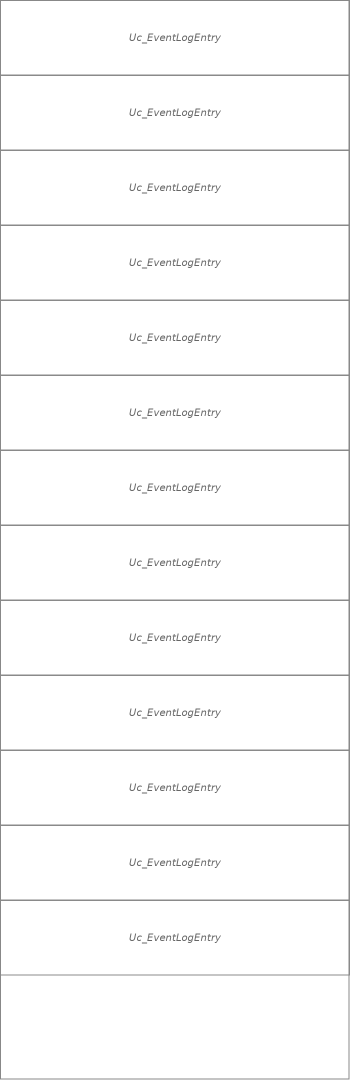
VISUALIZATION Uc_EventLogTable  // 350x1080
    Frame (0,0 350x75)
        shows Uc_EventLogEntry(stVisu := stVisu.astEvents[0], nSelectId := stVisu.nIdx, bQuit := stVisu.bQuitt)
    Frame (0,75 350x75)
        shows Uc_EventLogEntry(stVisu := stVisu.astEvents[1], nSelectId := stVisu.nIdx, bQuit := stVisu.bQuitt)
    Frame (0,150 350x75)
        shows Uc_EventLogEntry(stVisu := stVisu.astEvents[2], nSelectId := stVisu.nIdx, bQuit := stVisu.bQuitt)
    Frame (0,225 350x75)
        shows Uc_EventLogEntry(stVisu := stVisu.astEvents[3], nSelectId := stVisu.nIdx, bQuit := stVisu.bQuitt)
    Frame (0,300 350x75)
        shows Uc_EventLogEntry(stVisu := stVisu.astEvents[4], nSelectId := stVisu.nIdx, bQuit := stVisu.bQuitt)
    Frame (0,375 350x75)
        shows Uc_EventLogEntry(stVisu := stVisu.astEvents[5], nSelectId := stVisu.nIdx, bQuit := stVisu.bQuitt)
    Frame (0,450 350x75)
        shows Uc_EventLogEntry(stVisu := stVisu.astEvents[6], nSelectId := stVisu.nIdx, bQuit := stVisu.bQuitt)
    Frame (0,525 350x75)
        shows Uc_EventLogEntry(stVisu := stVisu.astEvents[7], nSelectId := stVisu.nIdx, bQuit := stVisu.bQuitt)
    Frame (0,600 350x75)
        shows Uc_EventLogEntry(stVisu := stVisu.astEvents[8], nSelectId := stVisu.nIdx, bQuit := stVisu.bQuitt)
    Frame (0,675 350x75)
        shows Uc_EventLogEntry(stVisu := stVisu.astEvents[9], nSelectId := stVisu.nIdx, bQuit := stVisu.bQuitt)
    Frame (0,750 350x75)
        shows Uc_EventLogEntry(stVisu := stVisu.astEvents[10], nSelectId := stVisu.nIdx, bQuit := stVisu.bQuitt)
    Frame (0,825 350x75)
        shows Uc_EventLogEntry(stVisu := stVisu.astEvents[11], nSelectId := stVisu.nIdx, bQuit := stVisu.bQuitt)
    Frame (0,900 350x75)
        shows Uc_EventLogEntry(stVisu := stVisu.astEvents[12], nSelectId := stVisu.nIdx, bQuit := stVisu.bQuitt)
END_VISUALIZATION

(* stored: Version 1.1.0.1
   Visu Uc_EventLogTable: Id {a7940e67-9a87-465f-a263-d9781aa5d3c9} *)
